Staubli VAL3: CloseAll.pgx

public program CloseAll()
begin
  dOut["dOut1"]=false
  dOut["dOut2"]=false
  dOut["dOut3"]=false
  dOut["dOut4"]=false
  dOut["dOut5"]=false
  dOut["dOut6"]=false
  dOut["dOut7"]=false
  dOut["dOut8"]=false
  dOut["dOut9"]=false
  dOut["dOut10"]=false
  dOut["dOut11"]=false
  dOut["dOut12"]=false
  dOut["dOut13"]=false
  dOut["dOut14"]=false
  dOut["dOut15"]=false
  dOut["dOut16"]=false
end
